TYPE ST_InfeedStatus :
	STRUCT
		ConveyorRunning : BOOL;
	END_STRUCT
END_TYPE

(* stored: Version 1.1.0.1, ProductVersion 3.1.4024.12
   DUT ST_InfeedStatus: Id {448395b4-4e11-452f-9da3-51f01c430932} *)
